Staubli VAL3: TrajSimu.pgx

public program TrajSimu(num x_nTrajIndex)
  local bool l_bRes
begin

  //路径模拟
  //需要读取文件

  //初始化
  call KillTask()
  //DataBase:bSimuIO=false
  DataBase:bIOStart=false
  nStartTraj=min(max(x_nTrajIndex,1),TxtFile:nTotalTraj)
  nEndTraj=min(TxtFile:nTotalTraj,x_nTrajIndex)


  //新建任务，来读写
  TxtFile:bReadProduct=true
  TxtFile:nReadCutCount=0
  taskCreate "ReadFile",100,ReadTraj()
  //taskCreateSync "Preset",0.008,bSync,Preset()
  taskCreate "Preset",100,Preset()
  if TxtFile:bWeldEnable
    //taskCreateSync "WeldEnd",0.008,bSync,WeldEnd()
  endIf

  //等待运动读写
  delay(0.5)
  //进行运动

  call Move()

end
